(* Schneider Machine Expert - Basic project Partida direta, file version 3.0.0.0 *)
(* ProjectInformations: Name=Partida Direta de Motor *)
(* UserInformations: LastName=Teodoro Araujo junior, FirstName=Sidney, CellNumber=27996489123, Email=sidneyteodoroaraujojunior2002@gmail.com, Street=Tupinambás, City=Belo Horizonte, ZipCode=30120040, State=Minas Gerais, Country=Brasil *)

HARDWARE
  Cpu 0: TM221CE24R
  EthernetConfiguration: NetworkName=M221, IpAllocationMode=FixedAddress, IpAddress=0.0.0.0, SubnetMask=0.0.0.0
  SerialLineConfiguration: Baud=Baud19200, Parity=ParityEven, DataBits=DataBits8, StopBits=StopBits1, PhysicalMedium=PhysicalMediumRs485, TransmissionMode=TransmissionModeModbusRtu, SlaveId=1, Addressing=SlaveAddressing
  MastTask: UsePeriodScanMode=false, PeriodScan=100
  FastTask: Period=255
  CpuBehavior: StartingMode=StartAsPreviousState, AutoSaveRamOnEeprom=true, WatchdogPeriod=250

SYMBOLS  (address, symbol, comment, settings)
  %I0.0     RELÉ  "Relé Térmico"
  %I0.1     OFF  "Desliga"
  %I0.2     ON  "Liga"
  %I0.3     STOP  "Botão de emergência"
  %Q0.0     MOTOR_0  "Motor"
  %Q0.1     H0  "Sinaleiro"
  %Q0.2     H1  "Sinaleiro"
  %Q0.3     H2  "Sinaleiro"
  %Q0.4     H3  "Sinaleiro"

POU Novo POU
  (* SectionNumber=1 *)

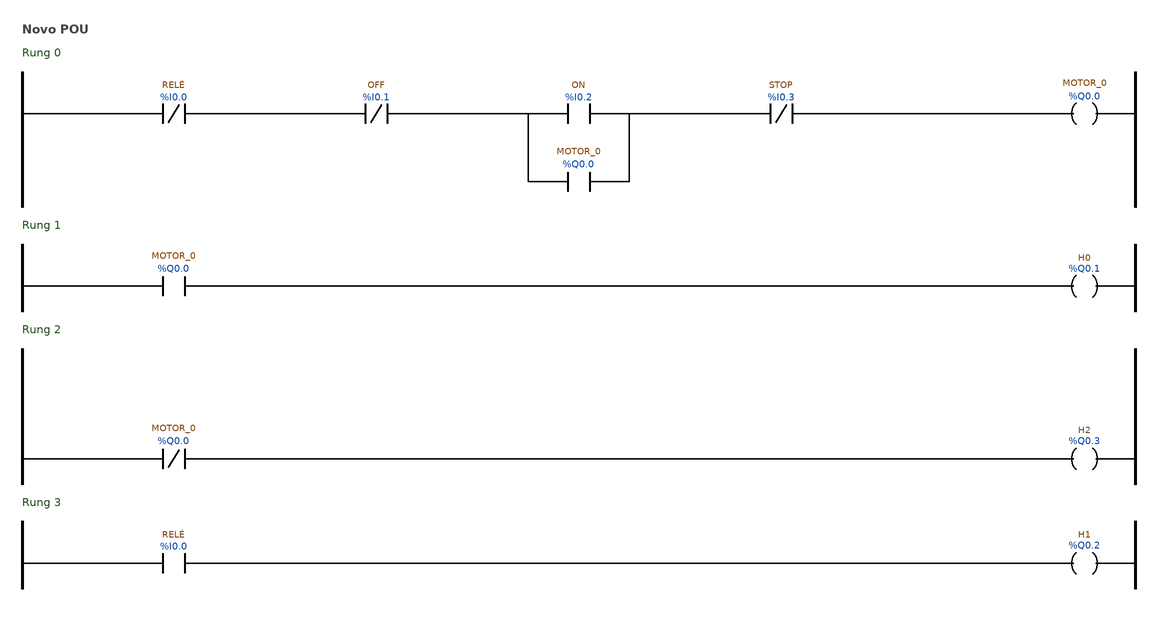

// Rung 0
  LDN %I0.0               (* RELÉ *)
  ANDN %I0.1              (* OFF *)
  AND( %I0.2              (* ON *)
  OR %Q0.0                (* MOTOR_0 *)
  )
  ANDN %I0.3              (* STOP *)
  ST %Q0.0                (* MOTOR_0 *)
  // as ST:
  //   MOTOR_0 := NOT RELÉ AND NOT OFF AND (ON OR MOTOR_0) AND NOT STOP;

// Rung 1
  LD %Q0.0                (* MOTOR_0 *)
  ST %Q0.1                (* H0 *)
  // as ST:
  //   H0 := MOTOR_0;

// Rung 2
  LDN %Q0.0               (* MOTOR_0 *)
  ST %Q0.3                (* H2 *)
  // as ST:
  //   H2 := NOT MOTOR_0;

// Rung 3
  LD %I0.0                (* RELÉ *)
  ST %Q0.2                (* H1 *)
  // as ST:
  //   H1 := RELÉ;
